// TIA Portal V19 export
TYPE "UDT_DIN"
   STRUCT
      "time" : Struct   // Delay setpoints
         on_set : Int := 0;   // Desired delay to set the memory switch
         off_set : Int := 0;   // Desired delay to reset the memory switch
         on_act : Int := 0;   // Counted delay to set the memory switch
         off_act : Int := 0;   // Counted delay to reset the memory switch
      END_STRUCT;
      setup : Struct   // Setup of switch
         polarity { S7_SetPoint := 'True'} : Bool := false;   // 0=normal polarity, 1=reverse polarity
         triggerversion { S7_SetPoint := 'True'} : Bool := false;   // 0=switch inactive for triggerring, 1=switch active for triggering
      END_STRUCT;
      faults : Struct   // Faults
         din { S7_SetPoint := 'True'} : "UDT_ALARMACKN";   // Digital switch fault
         fpreset : Bool := false;   // Faceplate reset for individual treatment
      END_STRUCT;
      sim : Struct   // Simulation
         cmdon : Bool := false;   // simulation on command
         cmdoff : Bool := false;   // simulation off command
         simulated : Bool := false;   // 0=simulation off, 1=simulation on
         cmdforce : Bool := false;   // force switch command
         cmdunforce : Bool := false;   // unforce switch command
         forced : Bool := false;   // 0=unforced, 1=forced
      END_STRUCT;
      status : Struct   // Status
         rawinput : Bool := false;   // Status of raw input
         processed : Bool := false;   // Status of input after polarity
         switch_active : Bool := false;   // Switch is Active after delay on
         alarm_monitor : Bool := false;   // Alarm is monitored
         fault : Bool := false;   // Fault is activated
      END_STRUCT;
   END_STRUCT;
END_TYPE
